FUNCTION_BLOCK Machine EXTENDS FB_PackML_BaseModule
VAR
	AX5000	  : FB_Component_BasicAxis := (Name := 'AX 5000 Axis');
	SoE_Reset : FB_ResetRoutine_SoEDrive;
END_VAR

// Automatically enables and disables HMI control based on the PackML mode
METHOD PROTECTED HMIPermissions

// This method is called cyclically by CyclicLogic()
AllowHMIControl(TRUE);
END_METHOD

// Basic module initialization logic
METHOD PROTECTED Initialize : BOOL;

// This method is called by CyclicLogic() as required
Initialize := FALSE;
CASE DescendantSequenceState OF
	0:
		RegisterComponent(AX5000);
		AX5000.ResetMethod		:= SoE_Reset;
		DescendantSequenceState := DescendantSequenceState + 10;

	10:
		IF SUPER^.Initialize() THEN
			DescendantSequenceState := DescendantSequenceState + 10;
		END_IF

	20:
		Initialize := TRUE;
END_CASE
END_METHOD

END_FUNCTION_BLOCK

(* stored: Version 1.1.0.1, ProductVersion 3.1.4026.12
   POU Machine: Id {cca3e28e-f3ae-4719-97b2-36656ead17e9}, SpecialFunc None
   Method HMIPermissions: Id {5df147cd-29e7-4bf7-b60b-30257e93fa20}
   Method Initialize: Id {56278613-2cb0-414c-bcba-44ebd2ccd3a2} *)
